	WY11701_00 AT  %MX11704.0 : BOOL; (*STN 4 CDA CYLINDER - OUT (-162Y2) *)
	WY11701_01 AT  %MX11704.1 : BOOL; (*STN 4 CDA CYLINDER - OUT (-162Y2) *)
	WY11701_02 AT  %MX11704.2 : BOOL; (*STN 4 CDA CYLINDER - OUT (-162Y2) *)
	WY11701_03 AT  %MX11704.3 : BOOL; (*STN 4 CDA CYLINDER - OUT (-162Y2) *)
	WY11701_04 AT  %MX11704.4 : BOOL; (*STN 4 CDA CYLINDER - OUT (-162Y2) *)
	WY11701_05 AT  %MX11704.5 : BOOL; (*STN 4 CDA CYLINDER - OUT (-162Y2) *)
	WY11701_06 AT  %MX11704.6 : BOOL; (*STN 4 CDA CYLINDER - OUT (-162Y2) *)
	WY11701_07 AT  %MX11704.7 : BOOL; (*STN 4 CDA CYLINDER - OUT (-162Y2) *)
	WY11701_08 AT  %MX11704.8 : BOOL; (*STN 4 CDA CYLINDER - OUT (-162Y2) *)
	WY11701_09 AT  %MX11704.9 : BOOL; (*STN 4 CDA CYLINDER - OUT (-162Y2) *)
	WY11701_10 AT  %MX11704.10 : BOOL; (*STN 4 CDA CYLINDER - OUT (-162Y2) *)
	WY11701_11 AT  %MX11704.11 : BOOL; (*STN 4 CDA CYLINDER - OUT (-162Y2) *)
	WY11701_12 AT  %MX11704.12 : BOOL; (*STN 4 CDA CYLINDER - OUT (-162Y2) *)
	WY11701_13 AT  %MX11704.13 : BOOL; (*STN 4 CDA CYLINDER - OUT (-162Y2) *)
	WY11701_14 AT  %MX11704.14 : BOOL; (*STN 4 CDA CYLINDER - OUT (-162Y2) *)
	WY11701_15 AT  %MX11704.15 : BOOL; (*STN 4 CDA CYLINDER - OUT (-162Y2) *)
	WY11701_16 AT  %MX11704.16 : BOOL; (*STN 4 CDA CYLINDER - OUT (-162Y2) *)
	WY11701_17 AT  %MX11704.17 : BOOL; (*STN 4 CDA CYLINDER - OUT (-162Y2) *)
	WY11701_18 AT  %MX11704.18 : BOOL; (*STN 4 CDA CYLINDER - OUT (-162Y2) *)
	WY11701_19 AT  %MX11704.19 : BOOL; (*STN 4 CDA CYLINDER - OUT (-162Y2) *)
	WY11701_20 AT  %MX11704.20 : BOOL; (*STN 4 CDA CYLINDER - OUT (-162Y2) *)
	WY11701_21 AT  %MX11704.21 : BOOL; (*STN 4 CDA CYLINDER - OUT (-162Y2) *)
	WY11701_22 AT  %MX11704.22 : BOOL; (*STN 4 CDA CYLINDER - OUT (-162Y2) *)
	WY11701_23 AT  %MX11704.23 : BOOL; (*STN 4 CDA CYLINDER - OUT (-162Y2) *)
	WY11701_24 AT  %MX11704.24 : BOOL; (*STN 4 CDA CYLINDER - OUT (-162Y2) *)
	WY11701_25 AT  %MX11704.25 : BOOL; (*STN 4 CDA CYLINDER - OUT (-162Y2) *)
	WY11701_26 AT  %MX11704.26 : BOOL; (*STN 4 CDA CYLINDER - OUT (-162Y2) *)
	WY11701_27 AT  %MX11704.27 : BOOL; (*STN 4 CDA CYLINDER - OUT (-162Y2) *)
	WY11701_28 AT  %MX11704.28 : BOOL; (*STN 4 CDA CYLINDER - OUT (-162Y2) *)
	WY11701_29 AT  %MX11704.29 : BOOL; (*STN 4 CDA CYLINDER - OUT (-162Y2) *)
	WY11701_30 AT  %MX11704.30 : BOOL; (*STN 4 CDA CYLINDER - OUT (-162Y2) *)
	WY11701_31 AT  %MX11704.31 : BOOL; (*STN 4 CDA CYLINDER - OUT (-162Y2) *)

	WY11702_00 AT  %MX11708.0 : BOOL; (*RAMP PUMP AV (-162Y3) *)
	WY11702_01 AT  %MX11708.1 : BOOL; (*RAMP PUMP AV (-162Y3) *)
	WY11702_02 AT  %MX11708.2 : BOOL; (*RAMP PUMP AV (-162Y3) *)
	WY11702_03 AT  %MX11708.3 : BOOL; (*RAMP PUMP AV (-162Y3) *)
	WY11702_04 AT  %MX11708.4 : BOOL; (*RAMP PUMP AV (-162Y3) *)
	WY11702_05 AT  %MX11708.5 : BOOL; (*RAMP PUMP AV (-162Y3) *)
	WY11702_06 AT  %MX11708.6 : BOOL; (*RAMP PUMP AV (-162Y3) *)
	WY11702_07 AT  %MX11708.7 : BOOL; (*RAMP PUMP AV (-162Y3) *)
	WY11702_08 AT  %MX11708.8 : BOOL; (*RAMP PUMP AV (-162Y3) *)
	WY11702_09 AT  %MX11708.9 : BOOL; (*RAMP PUMP AV (-162Y3) *)
	WY11702_10 AT  %MX11708.10 : BOOL; (*RAMP PUMP AV (-162Y3) *)
	WY11702_11 AT  %MX11708.11 : BOOL; (*RAMP PUMP AV (-162Y3) *)
	WY11702_12 AT  %MX11708.12 : BOOL; (*RAMP PUMP AV (-162Y3) *)
	WY11702_13 AT  %MX11708.13 : BOOL; (*RAMP PUMP AV (-162Y3) *)
	WY11702_14 AT  %MX11708.14 : BOOL; (*RAMP PUMP AV (-162Y3) *)
	WY11702_15 AT  %MX11708.15 : BOOL; (*RAMP PUMP AV (-162Y3) *)
	WY11702_16 AT  %MX11708.16 : BOOL; (*RAMP PUMP AV (-162Y3) *)
	WY11702_17 AT  %MX11708.17 : BOOL; (*RAMP PUMP AV (-162Y3) *)
	WY11702_18 AT  %MX11708.18 : BOOL; (*RAMP PUMP AV (-162Y3) *)
	WY11702_19 AT  %MX11708.19 : BOOL; (*RAMP PUMP AV (-162Y3) *)
	WY11702_20 AT  %MX11708.20 : BOOL; (*RAMP PUMP AV (-162Y3) *)
	WY11702_21 AT  %MX11708.21 : BOOL; (*RAMP PUMP AV (-162Y3) *)
	WY11702_22 AT  %MX11708.22 : BOOL; (*RAMP PUMP AV (-162Y3) *)
	WY11702_23 AT  %MX11708.23 : BOOL; (*RAMP PUMP AV (-162Y3) *)
	WY11702_24 AT  %MX11708.24 : BOOL; (*RAMP PUMP AV (-162Y3) *)
	WY11702_25 AT  %MX11708.25 : BOOL; (*RAMP PUMP AV (-162Y3) *)
	WY11702_26 AT  %MX11708.26 : BOOL; (*RAMP PUMP AV (-162Y3) *)
	WY11702_27 AT  %MX11708.27 : BOOL; (*RAMP PUMP AV (-162Y3) *)
	WY11702_28 AT  %MX11708.28 : BOOL; (*RAMP PUMP AV (-162Y3) *)
	WY11702_29 AT  %MX11708.29 : BOOL; (*RAMP PUMP AV (-162Y3) *)
	WY11702_30 AT  %MX11708.30 : BOOL; (*RAMP PUMP AV (-162Y3) *)
	WY11702_31 AT  %MX11708.31 : BOOL; (*RAMP PUMP AV (-162Y3) *)

	WY11703_00 AT  %MX11712.0 : BOOL; (*RESERVED *)
	WY11703_01 AT  %MX11712.1 : BOOL; (*RESERVED *)
	WY11703_02 AT  %MX11712.2 : BOOL; (*RESERVED *)
	WY11703_03 AT  %MX11712.3 : BOOL; (*RESERVED *)
	WY11703_04 AT  %MX11712.4 : BOOL; (*RESERVED *)
	WY11703_05 AT  %MX11712.5 : BOOL; (*RESERVED *)
	WY11703_06 AT  %MX11712.6 : BOOL; (*RESERVED *)
	WY11703_07 AT  %MX11712.7 : BOOL; (*RESERVED *)
	WY11703_08 AT  %MX11712.8 : BOOL; (*RESERVED *)
	WY11703_09 AT  %MX11712.9 : BOOL; (*RESERVED *)
	WY11703_10 AT  %MX11712.10 : BOOL; (*RESERVED *)
	WY11703_11 AT  %MX11712.11 : BOOL; (*RESERVED *)
	WY11703_12 AT  %MX11712.12 : BOOL; (*RESERVED *)
	WY11703_13 AT  %MX11712.13 : BOOL; (*RESERVED *)
	WY11703_14 AT  %MX11712.14 : BOOL; (*RESERVED *)
	WY11703_15 AT  %MX11712.15 : BOOL; (*RESERVED *)
	WY11703_16 AT  %MX11712.16 : BOOL; (*RESERVED *)
	WY11703_17 AT  %MX11712.17 : BOOL; (*RESERVED *)
	WY11703_18 AT  %MX11712.18 : BOOL; (*RESERVED *)
	WY11703_19 AT  %MX11712.19 : BOOL; (*RESERVED *)
	WY11703_20 AT  %MX11712.20 : BOOL; (*RESERVED *)
	WY11703_21 AT  %MX11712.21 : BOOL; (*RESERVED *)
	WY11703_22 AT  %MX11712.22 : BOOL; (*RESERVED *)
	WY11703_23 AT  %MX11712.23 : BOOL; (*RESERVED *)
	WY11703_24 AT  %MX11712.24 : BOOL; (*RESERVED *)
	WY11703_25 AT  %MX11712.25 : BOOL; (*RESERVED *)
	WY11703_26 AT  %MX11712.26 : BOOL; (*RESERVED *)
	WY11703_27 AT  %MX11712.27 : BOOL; (*RESERVED *)
	WY11703_28 AT  %MX11712.28 : BOOL; (*RESERVED *)
	WY11703_29 AT  %MX11712.29 : BOOL; (*RESERVED *)
	WY11703_30 AT  %MX11712.30 : BOOL; (*RESERVED *)
	WY11703_31 AT  %MX11712.31 : BOOL; (*RESERVED *)

	WY11704_00 AT  %MX11716.0 : BOOL; (*RESERVED *)
	WY11704_01 AT  %MX11716.1 : BOOL; (*RESERVED *)
	WY11704_02 AT  %MX11716.2 : BOOL; (*RESERVED *)
	WY11704_03 AT  %MX11716.3 : BOOL; (*RESERVED *)
	WY11704_04 AT  %MX11716.4 : BOOL; (*RESERVED *)
	WY11704_05 AT  %MX11716.5 : BOOL; (*RESERVED *)
	WY11704_06 AT  %MX11716.6 : BOOL; (*RESERVED *)
	WY11704_07 AT  %MX11716.7 : BOOL; (*RESERVED *)
	WY11704_08 AT  %MX11716.8 : BOOL; (*RESERVED *)
	WY11704_09 AT  %MX11716.9 : BOOL; (*RESERVED *)
	WY11704_10 AT  %MX11716.10 : BOOL; (*RESERVED *)
	WY11704_11 AT  %MX11716.11 : BOOL; (*RESERVED *)
	WY11704_12 AT  %MX11716.12 : BOOL; (*RESERVED *)
	WY11704_13 AT  %MX11716.13 : BOOL; (*RESERVED *)
	WY11704_14 AT  %MX11716.14 : BOOL; (*RESERVED *)
	WY11704_15 AT  %MX11716.15 : BOOL; (*RESERVED *)
	WY11704_16 AT  %MX11716.16 : BOOL; (*RESERVED *)
	WY11704_17 AT  %MX11716.17 : BOOL; (*RESERVED *)
	WY11704_18 AT  %MX11716.18 : BOOL; (*RESERVED *)
	WY11704_19 AT  %MX11716.19 : BOOL; (*RESERVED *)
	WY11704_20 AT  %MX11716.20 : BOOL; (*RESERVED *)
	WY11704_21 AT  %MX11716.21 : BOOL; (*RESERVED *)
	WY11704_22 AT  %MX11716.22 : BOOL; (*RESERVED *)
	WY11704_23 AT  %MX11716.23 : BOOL; (*RESERVED *)
	WY11704_24 AT  %MX11716.24 : BOOL; (*RESERVED *)
	WY11704_25 AT  %MX11716.25 : BOOL; (*RESERVED *)
	WY11704_26 AT  %MX11716.26 : BOOL; (*RESERVED *)
	WY11704_27 AT  %MX11716.27 : BOOL; (*RESERVED *)
	WY11704_28 AT  %MX11716.28 : BOOL; (*RESERVED *)
	WY11704_29 AT  %MX11716.29 : BOOL; (*RESERVED *)
	WY11704_30 AT  %MX11716.30 : BOOL; (*RESERVED *)
	WY11704_31 AT  %MX11716.31 : BOOL; (*RESERVED *)

	WY11705_00 AT  %MX11720.0 : BOOL; (*RESERVED *)
	WY11705_01 AT  %MX11720.1 : BOOL; (*RESERVED *)
	WY11705_02 AT  %MX11720.2 : BOOL; (*RESERVED *)
	WY11705_03 AT  %MX11720.3 : BOOL; (*RESERVED *)
	WY11705_04 AT  %MX11720.4 : BOOL; (*RESERVED *)
	WY11705_05 AT  %MX11720.5 : BOOL; (*RESERVED *)
	WY11705_06 AT  %MX11720.6 : BOOL; (*RESERVED *)
	WY11705_07 AT  %MX11720.7 : BOOL; (*RESERVED *)
	WY11705_08 AT  %MX11720.8 : BOOL; (*RESERVED *)
	WY11705_09 AT  %MX11720.9 : BOOL; (*RESERVED *)
	WY11705_10 AT  %MX11720.10 : BOOL; (*RESERVED *)
	WY11705_11 AT  %MX11720.11 : BOOL; (*RESERVED *)
	WY11705_12 AT  %MX11720.12 : BOOL; (*RESERVED *)
	WY11705_13 AT  %MX11720.13 : BOOL; (*RESERVED *)
	WY11705_14 AT  %MX11720.14 : BOOL; (*RESERVED *)
	WY11705_15 AT  %MX11720.15 : BOOL; (*RESERVED *)
	WY11705_16 AT  %MX11720.16 : BOOL; (*RESERVED *)
	WY11705_17 AT  %MX11720.17 : BOOL; (*RESERVED *)
	WY11705_18 AT  %MX11720.18 : BOOL; (*RESERVED *)
	WY11705_19 AT  %MX11720.19 : BOOL; (*RESERVED *)
	WY11705_20 AT  %MX11720.20 : BOOL; (*RESERVED *)
	WY11705_21 AT  %MX11720.21 : BOOL; (*RESERVED *)
	WY11705_22 AT  %MX11720.22 : BOOL; (*RESERVED *)
	WY11705_23 AT  %MX11720.23 : BOOL; (*RESERVED *)
	WY11705_24 AT  %MX11720.24 : BOOL; (*RESERVED *)
	WY11705_25 AT  %MX11720.25 : BOOL; (*RESERVED *)
	WY11705_26 AT  %MX11720.26 : BOOL; (*RESERVED *)
	WY11705_27 AT  %MX11720.27 : BOOL; (*RESERVED *)
	WY11705_28 AT  %MX11720.28 : BOOL; (*RESERVED *)
	WY11705_29 AT  %MX11720.29 : BOOL; (*RESERVED *)
	WY11705_30 AT  %MX11720.30 : BOOL; (*RESERVED *)
	WY11705_31 AT  %MX11720.31 : BOOL; (*RESERVED *)

	WY11706_00 AT  %MX11724.0 : BOOL; (*RESERVED *)
	WY11706_01 AT  %MX11724.1 : BOOL; (*RESERVED *)
	WY11706_02 AT  %MX11724.2 : BOOL; (*RESERVED *)
	WY11706_03 AT  %MX11724.3 : BOOL; (*RESERVED *)
	WY11706_04 AT  %MX11724.4 : BOOL; (*RESERVED *)
	WY11706_05 AT  %MX11724.5 : BOOL; (*RESERVED *)
	WY11706_06 AT  %MX11724.6 : BOOL; (*RESERVED *)
	WY11706_07 AT  %MX11724.7 : BOOL; (*RESERVED *)
	WY11706_08 AT  %MX11724.8 : BOOL; (*RESERVED *)
	WY11706_09 AT  %MX11724.9 : BOOL; (*RESERVED *)
	WY11706_10 AT  %MX11724.10 : BOOL; (*RESERVED *)
	WY11706_11 AT  %MX11724.11 : BOOL; (*RESERVED *)
	WY11706_12 AT  %MX11724.12 : BOOL; (*RESERVED *)
	WY11706_13 AT  %MX11724.13 : BOOL; (*RESERVED *)
	WY11706_14 AT  %MX11724.14 : BOOL; (*RESERVED *)
	WY11706_15 AT  %MX11724.15 : BOOL; (*RESERVED *)
	WY11706_16 AT  %MX11724.16 : BOOL; (*RESERVED *)
	WY11706_17 AT  %MX11724.17 : BOOL; (*RESERVED *)
	WY11706_18 AT  %MX11724.18 : BOOL; (*RESERVED *)
	WY11706_19 AT  %MX11724.19 : BOOL; (*RESERVED *)
	WY11706_20 AT  %MX11724.20 : BOOL; (*RESERVED *)
	WY11706_21 AT  %MX11724.21 : BOOL; (*RESERVED *)
	WY11706_22 AT  %MX11724.22 : BOOL; (*RESERVED *)
	WY11706_23 AT  %MX11724.23 : BOOL; (*RESERVED *)
	WY11706_24 AT  %MX11724.24 : BOOL; (*RESERVED *)
	WY11706_25 AT  %MX11724.25 : BOOL; (*RESERVED *)
	WY11706_26 AT  %MX11724.26 : BOOL; (*RESERVED *)
	WY11706_27 AT  %MX11724.27 : BOOL; (*RESERVED *)
	WY11706_28 AT  %MX11724.28 : BOOL; (*RESERVED *)
	WY11706_29 AT  %MX11724.29 : BOOL; (*RESERVED *)
	WY11706_30 AT  %MX11724.30 : BOOL; (*RESERVED *)
	WY11706_31 AT  %MX11724.31 : BOOL; (*RESERVED *)

	WY11707_00 AT  %MX11728.0 : BOOL; (*RESERVED *)
	WY11707_01 AT  %MX11728.1 : BOOL; (*RESERVED *)
	WY11707_02 AT  %MX11728.2 : BOOL; (*RESERVED *)
	WY11707_03 AT  %MX11728.3 : BOOL; (*RESERVED *)
	WY11707_04 AT  %MX11728.4 : BOOL; (*RESERVED *)
	WY11707_05 AT  %MX11728.5 : BOOL; (*RESERVED *)
	WY11707_06 AT  %MX11728.6 : BOOL; (*RESERVED *)
	WY11707_07 AT  %MX11728.7 : BOOL; (*RESERVED *)
	WY11707_08 AT  %MX11728.8 : BOOL; (*RESERVED *)
	WY11707_09 AT  %MX11728.9 : BOOL; (*RESERVED *)
	WY11707_10 AT  %MX11728.10 : BOOL; (*RESERVED *)
	WY11707_11 AT  %MX11728.11 : BOOL; (*RESERVED *)
	WY11707_12 AT  %MX11728.12 : BOOL; (*RESERVED *)
	WY11707_13 AT  %MX11728.13 : BOOL; (*RESERVED *)
	WY11707_14 AT  %MX11728.14 : BOOL; (*RESERVED *)
	WY11707_15 AT  %MX11728.15 : BOOL; (*RESERVED *)
	WY11707_16 AT  %MX11728.16 : BOOL; (*RESERVED *)
	WY11707_17 AT  %MX11728.17 : BOOL; (*RESERVED *)
	WY11707_18 AT  %MX11728.18 : BOOL; (*RESERVED *)
	WY11707_19 AT  %MX11728.19 : BOOL; (*RESERVED *)
	WY11707_20 AT  %MX11728.20 : BOOL; (*RESERVED *)
	WY11707_21 AT  %MX11728.21 : BOOL; (*RESERVED *)
	WY11707_22 AT  %MX11728.22 : BOOL; (*RESERVED *)
	WY11707_23 AT  %MX11728.23 : BOOL; (*RESERVED *)
	WY11707_24 AT  %MX11728.24 : BOOL; (*RESERVED *)
	WY11707_25 AT  %MX11728.25 : BOOL; (*RESERVED *)
	WY11707_26 AT  %MX11728.26 : BOOL; (*RESERVED *)
	WY11707_27 AT  %MX11728.27 : BOOL; (*RESERVED *)
	WY11707_28 AT  %MX11728.28 : BOOL; (*RESERVED *)
	WY11707_29 AT  %MX11728.29 : BOOL; (*RESERVED *)
	WY11707_30 AT  %MX11728.30 : BOOL; (*RESERVED *)
	WY11707_31 AT  %MX11728.31 : BOOL; (*RESERVED *)

	WY11708_00 AT  %MX11732.0 : BOOL; (*RESERVED *)
	WY11708_01 AT  %MX11732.1 : BOOL; (*RESERVED *)
	WY11708_02 AT  %MX11732.2 : BOOL; (*RESERVED *)
	WY11708_03 AT  %MX11732.3 : BOOL; (*RESERVED *)
	WY11708_04 AT  %MX11732.4 : BOOL; (*RESERVED *)
	WY11708_05 AT  %MX11732.5 : BOOL; (*RESERVED *)
	WY11708_06 AT  %MX11732.6 : BOOL; (*RESERVED *)
	WY11708_07 AT  %MX11732.7 : BOOL; (*RESERVED *)
	WY11708_08 AT  %MX11732.8 : BOOL; (*RESERVED *)
	WY11708_09 AT  %MX11732.9 : BOOL; (*RESERVED *)
	WY11708_10 AT  %MX11732.10 : BOOL; (*RESERVED *)
	WY11708_11 AT  %MX11732.11 : BOOL; (*RESERVED *)
	WY11708_12 AT  %MX11732.12 : BOOL; (*RESERVED *)
	WY11708_13 AT  %MX11732.13 : BOOL; (*RESERVED *)
	WY11708_14 AT  %MX11732.14 : BOOL; (*RESERVED *)
	WY11708_15 AT  %MX11732.15 : BOOL; (*RESERVED *)
	WY11708_16 AT  %MX11732.16 : BOOL; (*RESERVED *)
	WY11708_17 AT  %MX11732.17 : BOOL; (*RESERVED *)
	WY11708_18 AT  %MX11732.18 : BOOL; (*RESERVED *)
	WY11708_19 AT  %MX11732.19 : BOOL; (*RESERVED *)
	WY11708_20 AT  %MX11732.20 : BOOL; (*RESERVED *)
	WY11708_21 AT  %MX11732.21 : BOOL; (*RESERVED *)
	WY11708_22 AT  %MX11732.22 : BOOL; (*RESERVED *)
	WY11708_23 AT  %MX11732.23 : BOOL; (*RESERVED *)
	WY11708_24 AT  %MX11732.24 : BOOL; (*RESERVED *)
	WY11708_25 AT  %MX11732.25 : BOOL; (*RESERVED *)
	WY11708_26 AT  %MX11732.26 : BOOL; (*RESERVED *)
	WY11708_27 AT  %MX11732.27 : BOOL; (*RESERVED *)
	WY11708_28 AT  %MX11732.28 : BOOL; (*RESERVED *)
	WY11708_29 AT  %MX11732.29 : BOOL; (*RESERVED *)
	WY11708_30 AT  %MX11732.30 : BOOL; (*RESERVED *)
	WY11708_31 AT  %MX11732.31 : BOOL; (*RESERVED *)

	WY11709_00 AT  %MX11736.0 : BOOL; (*RESERVED *)
	WY11709_01 AT  %MX11736.1 : BOOL; (*RESERVED *)
	WY11709_02 AT  %MX11736.2 : BOOL; (*RESERVED *)
	WY11709_03 AT  %MX11736.3 : BOOL; (*RESERVED *)
	WY11709_04 AT  %MX11736.4 : BOOL; (*RESERVED *)
	WY11709_05 AT  %MX11736.5 : BOOL; (*RESERVED *)
	WY11709_06 AT  %MX11736.6 : BOOL; (*RESERVED *)
	WY11709_07 AT  %MX11736.7 : BOOL; (*RESERVED *)
	WY11709_08 AT  %MX11736.8 : BOOL; (*RESERVED *)
	WY11709_09 AT  %MX11736.9 : BOOL; (*RESERVED *)
	WY11709_10 AT  %MX11736.10 : BOOL; (*RESERVED *)
	WY11709_11 AT  %MX11736.11 : BOOL; (*RESERVED *)
	WY11709_12 AT  %MX11736.12 : BOOL; (*RESERVED *)
	WY11709_13 AT  %MX11736.13 : BOOL; (*RESERVED *)
	WY11709_14 AT  %MX11736.14 : BOOL; (*RESERVED *)
	WY11709_15 AT  %MX11736.15 : BOOL; (*RESERVED *)
	WY11709_16 AT  %MX11736.16 : BOOL; (*RESERVED *)
	WY11709_17 AT  %MX11736.17 : BOOL; (*RESERVED *)
	WY11709_18 AT  %MX11736.18 : BOOL; (*RESERVED *)
	WY11709_19 AT  %MX11736.19 : BOOL; (*RESERVED *)
	WY11709_20 AT  %MX11736.20 : BOOL; (*RESERVED *)
	WY11709_21 AT  %MX11736.21 : BOOL; (*RESERVED *)
	WY11709_22 AT  %MX11736.22 : BOOL; (*RESERVED *)
	WY11709_23 AT  %MX11736.23 : BOOL; (*RESERVED *)
	WY11709_24 AT  %MX11736.24 : BOOL; (*RESERVED *)
	WY11709_25 AT  %MX11736.25 : BOOL; (*RESERVED *)
	WY11709_26 AT  %MX11736.26 : BOOL; (*RESERVED *)
	WY11709_27 AT  %MX11736.27 : BOOL; (*RESERVED *)
	WY11709_28 AT  %MX11736.28 : BOOL; (*RESERVED *)
	WY11709_29 AT  %MX11736.29 : BOOL; (*RESERVED *)
	WY11709_30 AT  %MX11736.30 : BOOL; (*RESERVED *)
	WY11709_31 AT  %MX11736.31 : BOOL; (*RESERVED *)

	WY11710_00 AT  %MX11740.0 : BOOL; (*RESERVED *)
	WY11710_01 AT  %MX11740.1 : BOOL; (*RESERVED *)
	WY11710_02 AT  %MX11740.2 : BOOL; (*RESERVED *)
	WY11710_03 AT  %MX11740.3 : BOOL; (*RESERVED *)
	WY11710_04 AT  %MX11740.4 : BOOL; (*RESERVED *)
	WY11710_05 AT  %MX11740.5 : BOOL; (*RESERVED *)
	WY11710_06 AT  %MX11740.6 : BOOL; (*RESERVED *)
	WY11710_07 AT  %MX11740.7 : BOOL; (*RESERVED *)
	WY11710_08 AT  %MX11740.8 : BOOL; (*RESERVED *)
	WY11710_09 AT  %MX11740.9 : BOOL; (*RESERVED *)
	WY11710_10 AT  %MX11740.10 : BOOL; (*RESERVED *)
	WY11710_11 AT  %MX11740.11 : BOOL; (*RESERVED *)
	WY11710_12 AT  %MX11740.12 : BOOL; (*RESERVED *)
	WY11710_13 AT  %MX11740.13 : BOOL; (*RESERVED *)
	WY11710_14 AT  %MX11740.14 : BOOL; (*RESERVED *)
	WY11710_15 AT  %MX11740.15 : BOOL; (*RESERVED *)
	WY11710_16 AT  %MX11740.16 : BOOL; (*RESERVED *)
	WY11710_17 AT  %MX11740.17 : BOOL; (*RESERVED *)
	WY11710_18 AT  %MX11740.18 : BOOL; (*RESERVED *)
	WY11710_19 AT  %MX11740.19 : BOOL; (*RESERVED *)
	WY11710_20 AT  %MX11740.20 : BOOL; (*RESERVED *)
	WY11710_21 AT  %MX11740.21 : BOOL; (*RESERVED *)
	WY11710_22 AT  %MX11740.22 : BOOL; (*RESERVED *)
	WY11710_23 AT  %MX11740.23 : BOOL; (*RESERVED *)
	WY11710_24 AT  %MX11740.24 : BOOL; (*RESERVED *)
	WY11710_25 AT  %MX11740.25 : BOOL; (*RESERVED *)
	WY11710_26 AT  %MX11740.26 : BOOL; (*RESERVED *)
	WY11710_27 AT  %MX11740.27 : BOOL; (*RESERVED *)
	WY11710_28 AT  %MX11740.28 : BOOL; (*RESERVED *)
	WY11710_29 AT  %MX11740.29 : BOOL; (*RESERVED *)
	WY11710_30 AT  %MX11740.30 : BOOL; (*RESERVED *)
	WY11710_31 AT  %MX11740.31 : BOOL; (*RESERVED *)

	WY11711_00 AT  %MX11744.0 : BOOL; (*RESERVED *)
	WY11711_01 AT  %MX11744.1 : BOOL; (*RESERVED *)
	WY11711_02 AT  %MX11744.2 : BOOL; (*RESERVED *)
	WY11711_03 AT  %MX11744.3 : BOOL; (*RESERVED *)
	WY11711_04 AT  %MX11744.4 : BOOL; (*RESERVED *)
	WY11711_05 AT  %MX11744.5 : BOOL; (*RESERVED *)
	WY11711_06 AT  %MX11744.6 : BOOL; (*RESERVED *)
	WY11711_07 AT  %MX11744.7 : BOOL; (*RESERVED *)
	WY11711_08 AT  %MX11744.8 : BOOL; (*RESERVED *)
	WY11711_09 AT  %MX11744.9 : BOOL; (*RESERVED *)
	WY11711_10 AT  %MX11744.10 : BOOL; (*RESERVED *)
	WY11711_11 AT  %MX11744.11 : BOOL; (*RESERVED *)
	WY11711_12 AT  %MX11744.12 : BOOL; (*RESERVED *)
	WY11711_13 AT  %MX11744.13 : BOOL; (*RESERVED *)
	WY11711_14 AT  %MX11744.14 : BOOL; (*RESERVED *)
	WY11711_15 AT  %MX11744.15 : BOOL; (*RESERVED *)
	WY11711_16 AT  %MX11744.16 : BOOL; (*RESERVED *)
	WY11711_17 AT  %MX11744.17 : BOOL; (*RESERVED *)
	WY11711_18 AT  %MX11744.18 : BOOL; (*RESERVED *)
	WY11711_19 AT  %MX11744.19 : BOOL; (*RESERVED *)
	WY11711_20 AT  %MX11744.20 : BOOL; (*RESERVED *)
	WY11711_21 AT  %MX11744.21 : BOOL; (*RESERVED *)
	WY11711_22 AT  %MX11744.22 : BOOL; (*RESERVED *)
	WY11711_23 AT  %MX11744.23 : BOOL; (*RESERVED *)
	WY11711_24 AT  %MX11744.24 : BOOL; (*RESERVED *)
	WY11711_25 AT  %MX11744.25 : BOOL; (*RESERVED *)
	WY11711_26 AT  %MX11744.26 : BOOL; (*RESERVED *)
	WY11711_27 AT  %MX11744.27 : BOOL; (*RESERVED *)
	WY11711_28 AT  %MX11744.28 : BOOL; (*RESERVED *)
	WY11711_29 AT  %MX11744.29 : BOOL; (*RESERVED *)
	WY11711_30 AT  %MX11744.30 : BOOL; (*RESERVED *)
	WY11711_31 AT  %MX11744.31 : BOOL; (*RESERVED *)

	WY11712_00 AT  %MX11748.0 : BOOL; (*RESERVED *)
	WY11712_01 AT  %MX11748.1 : BOOL; (*RESERVED *)
	WY11712_02 AT  %MX11748.2 : BOOL; (*RESERVED *)
	WY11712_03 AT  %MX11748.3 : BOOL; (*RESERVED *)
	WY11712_04 AT  %MX11748.4 : BOOL; (*RESERVED *)
	WY11712_05 AT  %MX11748.5 : BOOL; (*RESERVED *)
	WY11712_06 AT  %MX11748.6 : BOOL; (*RESERVED *)
	WY11712_07 AT  %MX11748.7 : BOOL; (*RESERVED *)
	WY11712_08 AT  %MX11748.8 : BOOL; (*RESERVED *)
	WY11712_09 AT  %MX11748.9 : BOOL; (*RESERVED *)
	WY11712_10 AT  %MX11748.10 : BOOL; (*RESERVED *)
	WY11712_11 AT  %MX11748.11 : BOOL; (*RESERVED *)
	WY11712_12 AT  %MX11748.12 : BOOL; (*RESERVED *)
	WY11712_13 AT  %MX11748.13 : BOOL; (*RESERVED *)
	WY11712_14 AT  %MX11748.14 : BOOL; (*RESERVED *)
	WY11712_15 AT  %MX11748.15 : BOOL; (*RESERVED *)
	WY11712_16 AT  %MX11748.16 : BOOL; (*RESERVED *)
	WY11712_17 AT  %MX11748.17 : BOOL; (*RESERVED *)
	WY11712_18 AT  %MX11748.18 : BOOL; (*RESERVED *)
	WY11712_19 AT  %MX11748.19 : BOOL; (*RESERVED *)
	WY11712_20 AT  %MX11748.20 : BOOL; (*RESERVED *)
	WY11712_21 AT  %MX11748.21 : BOOL; (*RESERVED *)
	WY11712_22 AT  %MX11748.22 : BOOL; (*RESERVED *)
	WY11712_23 AT  %MX11748.23 : BOOL; (*RESERVED *)
	WY11712_24 AT  %MX11748.24 : BOOL; (*RESERVED *)
	WY11712_25 AT  %MX11748.25 : BOOL; (*RESERVED *)
	WY11712_26 AT  %MX11748.26 : BOOL; (*RESERVED *)
	WY11712_27 AT  %MX11748.27 : BOOL; (*RESERVED *)
	WY11712_28 AT  %MX11748.28 : BOOL; (*RESERVED *)
	WY11712_29 AT  %MX11748.29 : BOOL; (*RESERVED *)
	WY11712_30 AT  %MX11748.30 : BOOL; (*RESERVED *)
	WY11712_31 AT  %MX11748.31 : BOOL; (*RESERVED *)

	WY11713_00 AT  %MX11752.0 : BOOL; (*RESERVED *)
	WY11713_01 AT  %MX11752.1 : BOOL; (*RESERVED *)
	WY11713_02 AT  %MX11752.2 : BOOL; (*RESERVED *)
	WY11713_03 AT  %MX11752.3 : BOOL; (*RESERVED *)
	WY11713_04 AT  %MX11752.4 : BOOL; (*RESERVED *)
	WY11713_05 AT  %MX11752.5 : BOOL; (*RESERVED *)
	WY11713_06 AT  %MX11752.6 : BOOL; (*RESERVED *)
	WY11713_07 AT  %MX11752.7 : BOOL; (*RESERVED *)
	WY11713_08 AT  %MX11752.8 : BOOL; (*RESERVED *)
	WY11713_09 AT  %MX11752.9 : BOOL; (*RESERVED *)
	WY11713_10 AT  %MX11752.10 : BOOL; (*RESERVED *)
	WY11713_11 AT  %MX11752.11 : BOOL; (*RESERVED *)
	WY11713_12 AT  %MX11752.12 : BOOL; (*RESERVED *)
	WY11713_13 AT  %MX11752.13 : BOOL; (*RESERVED *)
	WY11713_14 AT  %MX11752.14 : BOOL; (*RESERVED *)
	WY11713_15 AT  %MX11752.15 : BOOL; (*RESERVED *)
	WY11713_16 AT  %MX11752.16 : BOOL; (*RESERVED *)
	WY11713_17 AT  %MX11752.17 : BOOL; (*RESERVED *)
	WY11713_18 AT  %MX11752.18 : BOOL; (*RESERVED *)
	WY11713_19 AT  %MX11752.19 : BOOL; (*RESERVED *)
	WY11713_20 AT  %MX11752.20 : BOOL; (*RESERVED *)
	WY11713_21 AT  %MX11752.21 : BOOL; (*RESERVED *)
	WY11713_22 AT  %MX11752.22 : BOOL; (*RESERVED *)
	WY11713_23 AT  %MX11752.23 : BOOL; (*RESERVED *)
	WY11713_24 AT  %MX11752.24 : BOOL; (*RESERVED *)
	WY11713_25 AT  %MX11752.25 : BOOL; (*RESERVED *)
	WY11713_26 AT  %MX11752.26 : BOOL; (*RESERVED *)
	WY11713_27 AT  %MX11752.27 : BOOL; (*RESERVED *)
	WY11713_28 AT  %MX11752.28 : BOOL; (*RESERVED *)
	WY11713_29 AT  %MX11752.29 : BOOL; (*RESERVED *)
	WY11713_30 AT  %MX11752.30 : BOOL; (*RESERVED *)
	WY11713_31 AT  %MX11752.31 : BOOL; (*RESERVED *)

	WY11714_00 AT  %MX11756.0 : BOOL; (*RESERVED *)
	WY11714_01 AT  %MX11756.1 : BOOL; (*RESERVED *)
	WY11714_02 AT  %MX11756.2 : BOOL; (*RESERVED *)
	WY11714_03 AT  %MX11756.3 : BOOL; (*RESERVED *)
	WY11714_04 AT  %MX11756.4 : BOOL; (*RESERVED *)
	WY11714_05 AT  %MX11756.5 : BOOL; (*RESERVED *)
	WY11714_06 AT  %MX11756.6 : BOOL; (*RESERVED *)
	WY11714_07 AT  %MX11756.7 : BOOL; (*RESERVED *)
	WY11714_08 AT  %MX11756.8 : BOOL; (*RESERVED *)
	WY11714_09 AT  %MX11756.9 : BOOL; (*RESERVED *)
	WY11714_10 AT  %MX11756.10 : BOOL; (*RESERVED *)
	WY11714_11 AT  %MX11756.11 : BOOL; (*RESERVED *)
	WY11714_12 AT  %MX11756.12 : BOOL; (*RESERVED *)
	WY11714_13 AT  %MX11756.13 : BOOL; (*RESERVED *)
	WY11714_14 AT  %MX11756.14 : BOOL; (*RESERVED *)
	WY11714_15 AT  %MX11756.15 : BOOL; (*RESERVED *)
	WY11714_16 AT  %MX11756.16 : BOOL; (*RESERVED *)
	WY11714_17 AT  %MX11756.17 : BOOL; (*RESERVED *)
	WY11714_18 AT  %MX11756.18 : BOOL; (*RESERVED *)
	WY11714_19 AT  %MX11756.19 : BOOL; (*RESERVED *)
	WY11714_20 AT  %MX11756.20 : BOOL; (*RESERVED *)
	WY11714_21 AT  %MX11756.21 : BOOL; (*RESERVED *)
	WY11714_22 AT  %MX11756.22 : BOOL; (*RESERVED *)
	WY11714_23 AT  %MX11756.23 : BOOL; (*RESERVED *)
	WY11714_24 AT  %MX11756.24 : BOOL; (*RESERVED *)
	WY11714_25 AT  %MX11756.25 : BOOL; (*RESERVED *)
	WY11714_26 AT  %MX11756.26 : BOOL; (*RESERVED *)
	WY11714_27 AT  %MX11756.27 : BOOL; (*RESERVED *)
	WY11714_28 AT  %MX11756.28 : BOOL; (*RESERVED *)
	WY11714_29 AT  %MX11756.29 : BOOL; (*RESERVED *)
	WY11714_30 AT  %MX11756.30 : BOOL; (*RESERVED *)
	WY11714_31 AT  %MX11756.31 : BOOL; (*RESERVED *)

	WY11715_00 AT  %MX11760.0 : BOOL; (*RESERVED *)
	WY11715_01 AT  %MX11760.1 : BOOL; (*RESERVED *)
	WY11715_02 AT  %MX11760.2 : BOOL; (*RESERVED *)
	WY11715_03 AT  %MX11760.3 : BOOL; (*RESERVED *)
	WY11715_04 AT  %MX11760.4 : BOOL; (*RESERVED *)
	WY11715_05 AT  %MX11760.5 : BOOL; (*RESERVED *)
	WY11715_06 AT  %MX11760.6 : BOOL; (*RESERVED *)
	WY11715_07 AT  %MX11760.7 : BOOL; (*RESERVED *)
	WY11715_08 AT  %MX11760.8 : BOOL; (*RESERVED *)
	WY11715_09 AT  %MX11760.9 : BOOL; (*RESERVED *)
	WY11715_10 AT  %MX11760.10 : BOOL; (*RESERVED *)
	WY11715_11 AT  %MX11760.11 : BOOL; (*RESERVED *)
	WY11715_12 AT  %MX11760.12 : BOOL; (*RESERVED *)
	WY11715_13 AT  %MX11760.13 : BOOL; (*RESERVED *)
	WY11715_14 AT  %MX11760.14 : BOOL; (*RESERVED *)
	WY11715_15 AT  %MX11760.15 : BOOL; (*RESERVED *)
	WY11715_16 AT  %MX11760.16 : BOOL; (*RESERVED *)
	WY11715_17 AT  %MX11760.17 : BOOL; (*RESERVED *)
	WY11715_18 AT  %MX11760.18 : BOOL; (*RESERVED *)
	WY11715_19 AT  %MX11760.19 : BOOL; (*RESERVED *)
	WY11715_20 AT  %MX11760.20 : BOOL; (*RESERVED *)
	WY11715_21 AT  %MX11760.21 : BOOL; (*RESERVED *)
	WY11715_22 AT  %MX11760.22 : BOOL; (*RESERVED *)
	WY11715_23 AT  %MX11760.23 : BOOL; (*RESERVED *)
	WY11715_24 AT  %MX11760.24 : BOOL; (*RESERVED *)
	WY11715_25 AT  %MX11760.25 : BOOL; (*RESERVED *)
	WY11715_26 AT  %MX11760.26 : BOOL; (*RESERVED *)
	WY11715_27 AT  %MX11760.27 : BOOL; (*RESERVED *)
	WY11715_28 AT  %MX11760.28 : BOOL; (*RESERVED *)
	WY11715_29 AT  %MX11760.29 : BOOL; (*RESERVED *)
	WY11715_30 AT  %MX11760.30 : BOOL; (*RESERVED *)
	WY11715_31 AT  %MX11760.31 : BOOL; (*RESERVED *)

END_VAR

(* stored: Version 1.1.0.1, ProductVersion 3.1.4024.12
   GVL Global_Variables_DigitalBoolCtrl: Id {aedac326-3064-4457-9efa-d4ee7b4885d2} *)
